FUNCTION_BLOCK farberkennung_HMI (* Service Interface Function Block Type *)
  (* Standard: 61499-2 *)
  (* Version 0.0, 12/04/2022, labor, Schneider Electric, template *)
  PACKAGE Main;
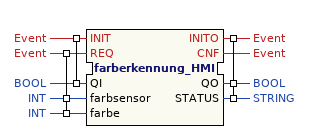
  EVENT_INPUT
    INIT WITH QI;
    REQ WITH farbsensor, farbe;
  END_EVENT
  EVENT_OUTPUT
    INITO WITH QO, STATUS;
    CNF;
  END_EVENT
  VAR_INPUT
    QI : BOOL;
    farbsensor : INT;
    farbe : INT;
  END_VAR
  VAR_OUTPUT
    QO : BOOL; (* Event Output Qualifier *)
    STATUS : STRING; (* Service Status *)
  END_VAR
  SERVICE /
    SEQUENCE 
    END_SEQUENCE
  END_SERVICE
END_FUNCTION_BLOCK
